// TIA Portal V19 export
DATA_BLOCK "Tor"   // DB1092
// stored: AutoNumber false, InstanceOfName RT, InstanceOfType FB
"RT"
   // VAR RETAIN
   //    In { ExternalAccessible := 'False'; ExternalVisible := 'False'; ExternalWritable := 'False'} : Struct
   //       NotHalt : Bool;
   //       MSS_ok : Bool;
   //       ok : Bool;
   //       Knauf_Auto : Bool;
   //       T_auf : Bool;
   //       T_zu : Bool;
   //       S_auf : Bool;
   //       S_zu : Bool;
   //       ErrQ : Bool;
   //       Sperrluft_ok : Bool;
   //       Kein_Gas_Alarm : Bool;
   //    END_STRUCT;
   //    Param { ExternalAccessible := 'False'; ExternalVisible := 'False'; ExternalWritable := 'False'} : Struct
   //       "TO" : Time;
   //    END_STRUCT;
   //    Zst { ExternalAccessible := 'False'; ExternalVisible := 'False'; ExternalWritable := 'False'} : Struct
   //       Req_Auf : Bool;
   //       Fehler : Bool;
   //       Sperre_QF : Bool;
   //       QF_sicher : Bool;
   //    END_STRUCT;
   //    Out { ExternalAccessible := 'False'; ExternalVisible := 'False'; ExternalWritable := 'False'} : Struct
   //       auf : Bool;
   //       zu : Bool;
   //    END_STRUCT;
   //    Mld { ExternalAccessible := 'False'; ExternalVisible := 'False'; ExternalWritable := 'False'} : Struct
   //       n_Auto : Bool;
   //       TO_auf : Bool;
   //       TO_zu : Bool;
   //       MSS : Bool;
   //       nok : Bool;
   //    END_STRUCT;
   // END_VAR
   // VAR
   //    IEC_Timer { ExternalAccessible := 'False'; ExternalVisible := 'False'; ExternalWritable := 'False'} : Struct
   //       TO_auf : TON_TIME;
   //       TO_zu : TON_TIME;
   //    END_STRUCT;
   // END_VAR
BEGIN
END_DATA_BLOCK
